// TIA Portal V17 export
// export: Created 2025-03-13T10:29:36.6380281Z, ExportSetting WithDefaults, DisplayName Totally Integrated Automation Portal, DisplayVersion V17 Update 8, DisplayName TIA Portal Openness, DisplayVersion V17 Update 8, DisplayName TIA Portal Version Control Interface, DisplayVersion V17, DisplayName SINAMICS Startdrive Advanced, DisplayVersion V17 SP2, DisplayName SINAMICS Startdrive G110M, G120, G120C, G120D, G120P, G115D, DisplayVersion V17 SP2, DisplayName SINAMICS Startdrive G130, G150, S120, S150, SINAMICS MV, S210, DisplayVersion V17 SP2, DisplayName STEP 7 Professional, DisplayVersion V17 Update 8, DisplayName SINUMERIK ONE STEP 7 Toolbox, DisplayVersion V17 Update 12, DisplayName SINUMERIK 840D sl STEP 7 Toolbox, DisplayVersion V17 Update 12, DisplayName STEP 7 Safety, DisplayVersion V17 Update 6, DisplayName WinCC Advanced, DisplayVersion V17 Update 8
FUNCTION_BLOCK "FB20300_LASER_GUIDE"   // FB20300, LAD
TITLE = FB20300 LASER GUIDE
{ S7_Optimized_Access := 'FALSE' }
VERSION : 0.1
// stored: AutoNumber false, IsIECCheckEnabled false, SetENOAutomatically false, UDAEnableTagReadback false
   VAR_INPUT
      iCONTROL_ON_DELAYED : Bool;
      iLASER_ACTIVE_LASER_ON : Bool;
      iSTART_MANUAL_REQUEST : Bool;
      iSTART_AUTO_REQUEST : Bool;
      iGUIDE_LASER_IS_ON : Bool;
      iSTOP_MANUAL_REQUEST : Bool;
      iSTOP_AUTO_REQUEST : Bool;
      iHOME_SEQUENCE_RUNNING : Bool;
      iCONTROL_OFF : Bool;
      TEMP : Timer;
   END_VAR
   VAR_OUTPUT
      oLASER_NOT_READY_ALARM : Bool;
      oSEOC_ALARMS : Bool;
      oSwitchoncondition_on : Bool;
      oSwitchoncondition_off : Bool;
      oMotion_Active_Right : Bool;
      oMotion_Active_Left : Bool;
      oLimit_right : Bool;
      oLimit_left : Bool;
      oGUIDE_LASER_ON : Bool;
   END_VAR
   VAR DB_SPECIFIC
      DATA : "LASER GUIDE";
   END_VAR
   VAR_TEMP
      DB_NUMBER : DInt;
   END_VAR
   VAR_TEMP   // added for the SCL form of the ladder/FBD networks
      _w1 : Bool;
      _s5time1 : S5Time;
   END_VAR
BEGIN

NETWORK
TITLE = READ INSTANCE DB NUMBER
      L     DINO;
      +     10#800000;
      T     #DB_NUMBER;

REGION Network 2: START GENERAL CONDITIONS / Start General Conditions
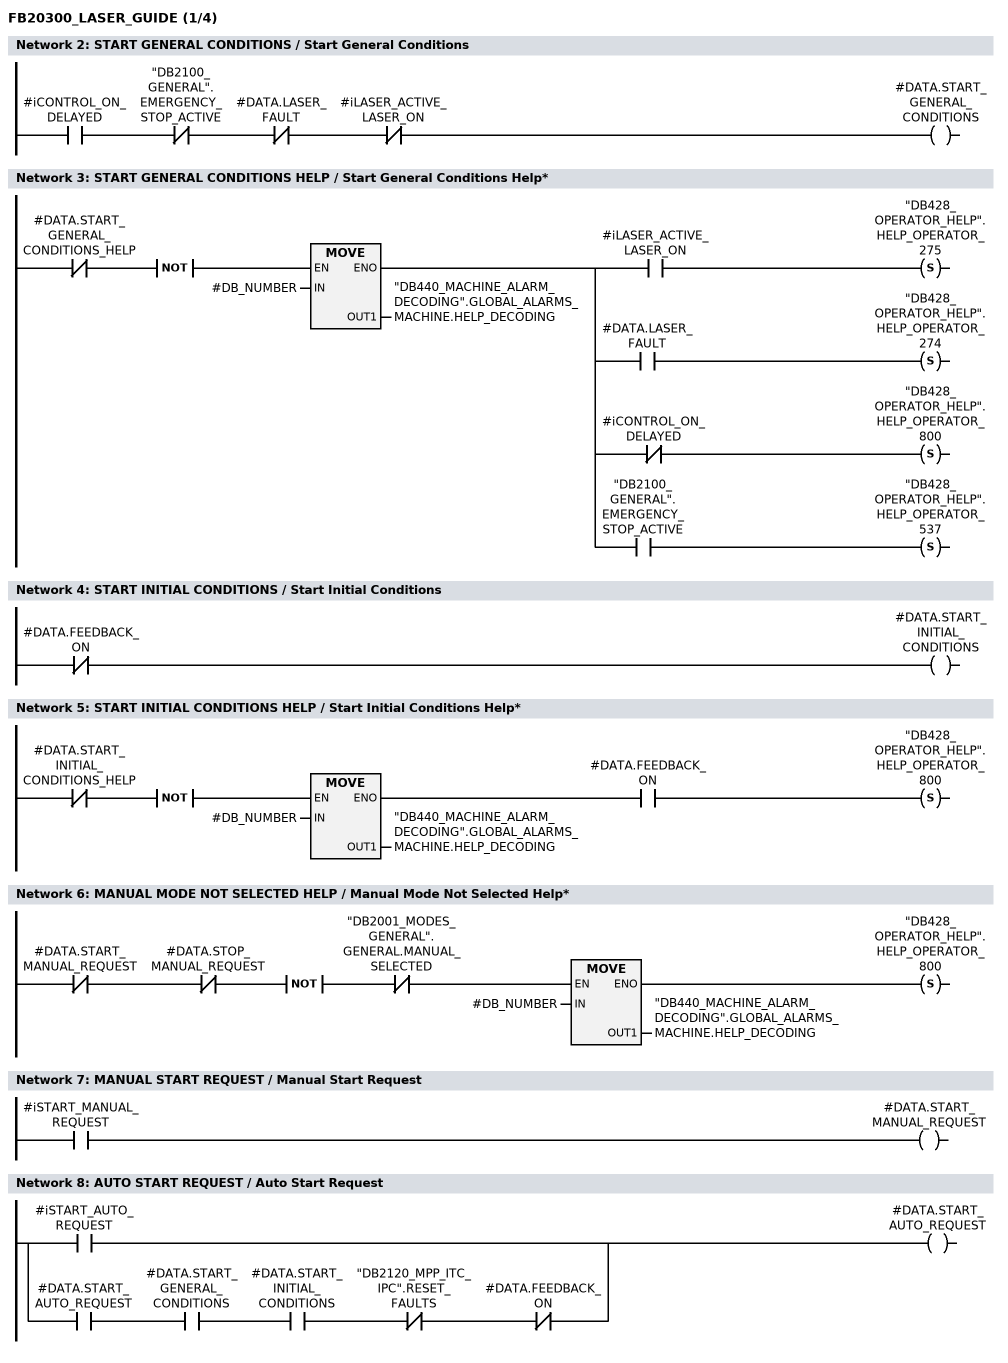
   RUNG wire#powerrail
      Contact( #iCONTROL_ON_DELAYED )
      I_Contact( "DB2100_GENERAL".EMERGENCY_STOP_ACTIVE )
      I_Contact( #DATA.LASER_FAULT )
      I_Contact( #iLASER_ACTIVE_LASER_ON )
      Coil( #DATA.START_GENERAL_CONDITIONS )
   END_RUNG
   // the same network as SCL:
   #DATA.START_GENERAL_CONDITIONS := #iCONTROL_ON_DELAYED AND NOT "DB2100_GENERAL".EMERGENCY_STOP_ACTIVE AND NOT #DATA.LASER_FAULT AND NOT #iLASER_ACTIVE_LASER_ON;
END_REGION

REGION Network 3: START GENERAL CONDITIONS HELP / Start General Conditions Help*
   RUNG wire#powerrail
      I_Contact( #DATA.START_GENERAL_CONDITIONS_HELP )
      Not()
      Move(in := #DB_NUMBER, out1 => "DB440_MACHINE_ALARM_DECODING".GLOBAL_ALARMS_MACHINE.HELP_DECODING)
      wire#w1
      Contact( #iLASER_ACTIVE_LASER_ON )
      S_Coil( "DB428_OPERATOR_HELP".HELP_OPERATOR_275 )
   END_RUNG
   RUNG wire#w1
      Contact( #DATA.LASER_FAULT )
      S_Coil( "DB428_OPERATOR_HELP".HELP_OPERATOR_274 )
   END_RUNG
   RUNG wire#w1
      I_Contact( #iCONTROL_ON_DELAYED )
      S_Coil( "DB428_OPERATOR_HELP".HELP_OPERATOR_800 )
   END_RUNG
   RUNG wire#w1
      Contact( "DB2100_GENERAL".EMERGENCY_STOP_ACTIVE )
      S_Coil( "DB428_OPERATOR_HELP".HELP_OPERATOR_537 )
   END_RUNG
   // the same network as SCL:
   #_w1 := NOT (NOT #DATA.START_GENERAL_CONDITIONS_HELP);
   IF #_w1 THEN "DB440_MACHINE_ALARM_DECODING".GLOBAL_ALARMS_MACHINE.HELP_DECODING := #DB_NUMBER; END_IF;
   IF #_w1 AND #iLASER_ACTIVE_LASER_ON THEN "DB428_OPERATOR_HELP".HELP_OPERATOR_275 := TRUE; END_IF;
   IF #_w1 AND #DATA.LASER_FAULT THEN "DB428_OPERATOR_HELP".HELP_OPERATOR_274 := TRUE; END_IF;
   IF #_w1 AND NOT #iCONTROL_ON_DELAYED THEN "DB428_OPERATOR_HELP".HELP_OPERATOR_800 := TRUE; END_IF;
   IF #_w1 AND "DB2100_GENERAL".EMERGENCY_STOP_ACTIVE THEN
       "DB428_OPERATOR_HELP".HELP_OPERATOR_537 := TRUE;
   END_IF;
END_REGION

REGION Network 4: START INITIAL CONDITIONS / Start Initial Conditions
   RUNG wire#powerrail
      I_Contact( #DATA.FEEDBACK_ON )
      Coil( #DATA.START_INITIAL_CONDITIONS )
   END_RUNG
   // the same network as SCL:
   #DATA.START_INITIAL_CONDITIONS := NOT #DATA.FEEDBACK_ON;
END_REGION

REGION Network 5: START INITIAL CONDITIONS HELP / Start Initial Conditions Help*
   RUNG wire#powerrail
      I_Contact( #DATA.START_INITIAL_CONDITIONS_HELP )
      Not()
      Move(in := #DB_NUMBER, out1 => "DB440_MACHINE_ALARM_DECODING".GLOBAL_ALARMS_MACHINE.HELP_DECODING)
      Contact( #DATA.FEEDBACK_ON )
      S_Coil( "DB428_OPERATOR_HELP".HELP_OPERATOR_800 )
   END_RUNG
   // the same network as SCL:
   #_w1 := NOT (NOT #DATA.START_INITIAL_CONDITIONS_HELP);
   IF #_w1 THEN "DB440_MACHINE_ALARM_DECODING".GLOBAL_ALARMS_MACHINE.HELP_DECODING := #DB_NUMBER; END_IF;
   IF #_w1 AND #DATA.FEEDBACK_ON THEN "DB428_OPERATOR_HELP".HELP_OPERATOR_800 := TRUE; END_IF;
END_REGION

REGION Network 6: MANUAL MODE NOT SELECTED HELP / Manual Mode Not Selected Help*
   RUNG wire#powerrail
      I_Contact( #DATA.START_MANUAL_REQUEST )
      I_Contact( #DATA.STOP_MANUAL_REQUEST )
      Not()
      I_Contact( "DB2001_MODES_GENERAL".GENERAL.MANUAL_SELECTED )
      Move(in := #DB_NUMBER, out1 => "DB440_MACHINE_ALARM_DECODING".GLOBAL_ALARMS_MACHINE.HELP_DECODING)
      S_Coil( "DB428_OPERATOR_HELP".HELP_OPERATOR_800 )
   END_RUNG
   // the same network as SCL:
   IF NOT (NOT #DATA.START_MANUAL_REQUEST AND NOT #DATA.STOP_MANUAL_REQUEST) AND NOT "DB2001_MODES_GENERAL".GENERAL.MANUAL_SELECTED THEN
       "DB440_MACHINE_ALARM_DECODING".GLOBAL_ALARMS_MACHINE.HELP_DECODING := #DB_NUMBER;
       "DB428_OPERATOR_HELP".HELP_OPERATOR_800 := TRUE;
   END_IF;
END_REGION

REGION Network 7: MANUAL START REQUEST / Manual Start Request
   RUNG wire#powerrail
      Contact( #iSTART_MANUAL_REQUEST )
      Coil( #DATA.START_MANUAL_REQUEST )
   END_RUNG
   // the same network as SCL:
   #DATA.START_MANUAL_REQUEST := #iSTART_MANUAL_REQUEST;
END_REGION

REGION Network 8: AUTO START REQUEST / Auto Start Request
   RUNG wire#powerrail
      Contact( #iSTART_AUTO_REQUEST )
      wire#w1
      Coil( #DATA.START_AUTO_REQUEST )
   END_RUNG
   RUNG wire#powerrail
      Contact( #DATA.START_AUTO_REQUEST )
      Contact( #DATA.START_GENERAL_CONDITIONS )
      Contact( #DATA.START_INITIAL_CONDITIONS )
      I_Contact( "DB2120_MPP_ITC_IPC".RESET_FAULTS )
      I_Contact( #DATA.FEEDBACK_ON )
   END_RUNG wire#w1
   // the same network as SCL:
   #DATA.START_AUTO_REQUEST := #iSTART_AUTO_REQUEST OR (#DATA.START_AUTO_REQUEST AND #DATA.START_GENERAL_CONDITIONS AND #DATA.START_INITIAL_CONDITIONS AND NOT "DB2120_MPP_ITC_IPC".RESET_FAULTS AND NOT #DATA.FEEDBACK_ON);
END_REGION

REGION Network 9: START GLOBAL REQUEST / Start Global Request / GLOBAL START REQUEST
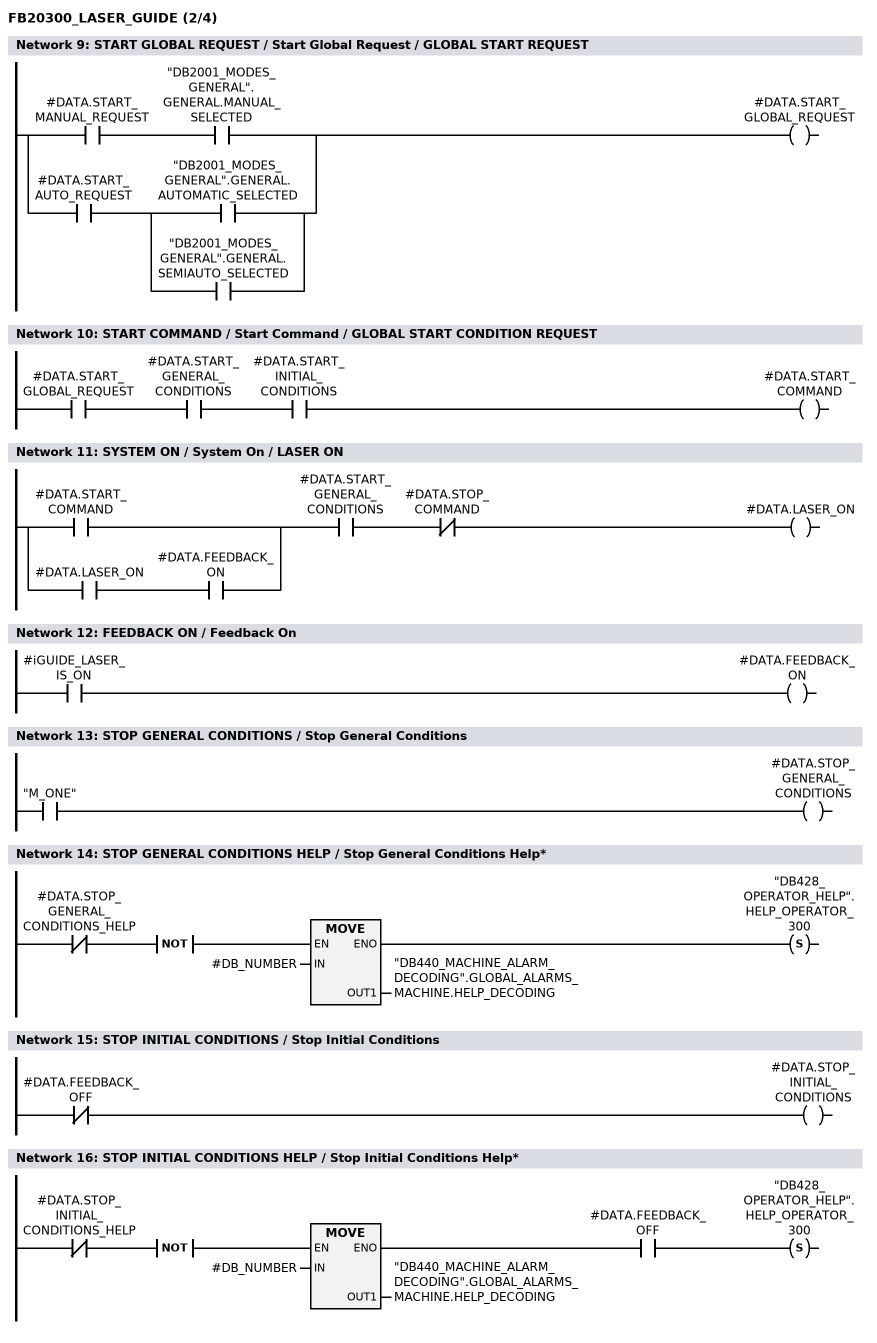
   RUNG wire#powerrail
      Contact( #DATA.START_MANUAL_REQUEST )
      Contact( "DB2001_MODES_GENERAL".GENERAL.MANUAL_SELECTED )
      wire#w1
      Coil( #DATA.START_GLOBAL_REQUEST )
   END_RUNG
   RUNG wire#powerrail
      Contact( #DATA.START_AUTO_REQUEST )
      wire#w2
      Contact( "DB2001_MODES_GENERAL".GENERAL.AUTOMATIC_SELECTED )
   END_RUNG wire#w1
   RUNG wire#w2
      Contact( "DB2001_MODES_GENERAL".GENERAL.SEMIAUTO_SELECTED )
   END_RUNG wire#w1
   // the same network as SCL:
   #DATA.START_GLOBAL_REQUEST := (#DATA.START_MANUAL_REQUEST AND "DB2001_MODES_GENERAL".GENERAL.MANUAL_SELECTED) OR (#DATA.START_AUTO_REQUEST AND ("DB2001_MODES_GENERAL".GENERAL.AUTOMATIC_SELECTED OR "DB2001_MODES_GENERAL".GENERAL.SEMIAUTO_SELECTED));
END_REGION

REGION Network 10: START COMMAND / Start Command / GLOBAL START CONDITION REQUEST
   RUNG wire#powerrail
      Contact( #DATA.START_GLOBAL_REQUEST )
      Contact( #DATA.START_GENERAL_CONDITIONS )
      Contact( #DATA.START_INITIAL_CONDITIONS )
      Coil( #DATA.START_COMMAND )
   END_RUNG
   // the same network as SCL:
   #DATA.START_COMMAND := #DATA.START_GLOBAL_REQUEST AND #DATA.START_GENERAL_CONDITIONS AND #DATA.START_INITIAL_CONDITIONS;
END_REGION

REGION Network 11: SYSTEM ON / System On / LASER ON
   RUNG wire#powerrail
      Contact( #DATA.START_COMMAND )
      wire#w1
      Contact( #DATA.START_GENERAL_CONDITIONS )
      I_Contact( #DATA.STOP_COMMAND )
      Coil( #DATA.LASER_ON )
   END_RUNG
   RUNG wire#powerrail
      Contact( #DATA.LASER_ON )
      Contact( #DATA.FEEDBACK_ON )
   END_RUNG wire#w1
   // the same network as SCL:
   #DATA.LASER_ON := (#DATA.START_COMMAND OR (#DATA.LASER_ON AND #DATA.FEEDBACK_ON)) AND #DATA.START_GENERAL_CONDITIONS AND NOT #DATA.STOP_COMMAND;
END_REGION

REGION Network 12: FEEDBACK ON / Feedback On
   RUNG wire#powerrail
      Contact( #iGUIDE_LASER_IS_ON )
      Coil( #DATA.FEEDBACK_ON )
   END_RUNG
   // the same network as SCL:
   #DATA.FEEDBACK_ON := #iGUIDE_LASER_IS_ON;
END_REGION

REGION Network 13: STOP GENERAL CONDITIONS / Stop General Conditions
   RUNG wire#powerrail
      Contact( "M_ONE" )
      Coil( #DATA.STOP_GENERAL_CONDITIONS )
   END_RUNG
   // the same network as SCL:
   #DATA.STOP_GENERAL_CONDITIONS := "M_ONE";
END_REGION

REGION Network 14: STOP GENERAL CONDITIONS HELP / Stop General Conditions Help*
   RUNG wire#powerrail
      I_Contact( #DATA.STOP_GENERAL_CONDITIONS_HELP )
      Not()
      Move(in := #DB_NUMBER, out1 => "DB440_MACHINE_ALARM_DECODING".GLOBAL_ALARMS_MACHINE.HELP_DECODING)
      S_Coil( "DB428_OPERATOR_HELP".HELP_OPERATOR_300 )
   END_RUNG
   // the same network as SCL:
   IF NOT (NOT #DATA.STOP_GENERAL_CONDITIONS_HELP) THEN
       "DB440_MACHINE_ALARM_DECODING".GLOBAL_ALARMS_MACHINE.HELP_DECODING := #DB_NUMBER;
       "DB428_OPERATOR_HELP".HELP_OPERATOR_300 := TRUE;
   END_IF;
END_REGION

REGION Network 15: STOP INITIAL CONDITIONS / Stop Initial Conditions
   RUNG wire#powerrail
      I_Contact( #DATA.FEEDBACK_OFF )
      Coil( #DATA.STOP_INITIAL_CONDITIONS )
   END_RUNG
   // the same network as SCL:
   #DATA.STOP_INITIAL_CONDITIONS := NOT #DATA.FEEDBACK_OFF;
END_REGION

REGION Network 16: STOP INITIAL CONDITIONS HELP / Stop Initial Conditions Help*
   RUNG wire#powerrail
      I_Contact( #DATA.STOP_INITIAL_CONDITIONS_HELP )
      Not()
      Move(in := #DB_NUMBER, out1 => "DB440_MACHINE_ALARM_DECODING".GLOBAL_ALARMS_MACHINE.HELP_DECODING)
      Contact( #DATA.FEEDBACK_OFF )
      S_Coil( "DB428_OPERATOR_HELP".HELP_OPERATOR_300 )
   END_RUNG
   // the same network as SCL:
   #_w1 := NOT (NOT #DATA.STOP_INITIAL_CONDITIONS_HELP);
   IF #_w1 THEN "DB440_MACHINE_ALARM_DECODING".GLOBAL_ALARMS_MACHINE.HELP_DECODING := #DB_NUMBER; END_IF;
   IF #_w1 AND #DATA.FEEDBACK_OFF THEN "DB428_OPERATOR_HELP".HELP_OPERATOR_300 := TRUE; END_IF;
END_REGION

REGION Network 17: MANUAL STOP REQUEST / Manual Stop Request
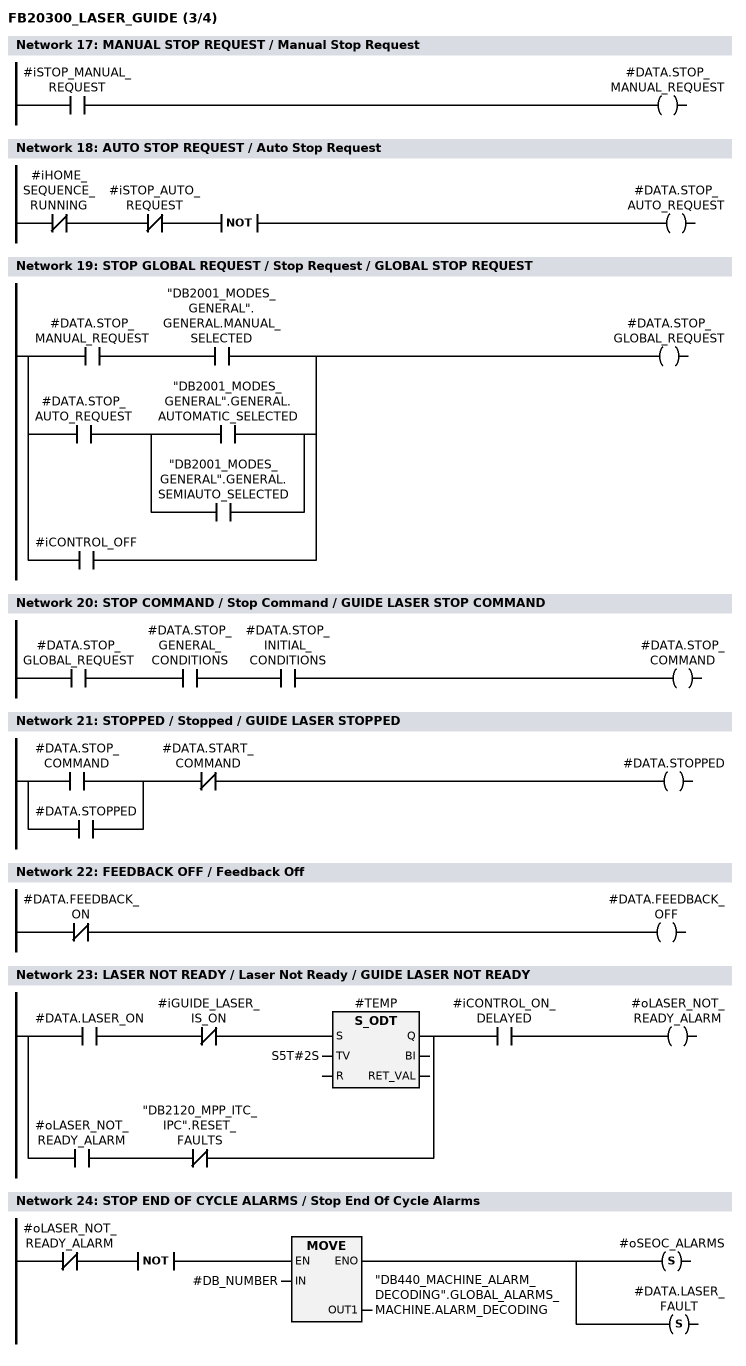
   RUNG wire#powerrail
      Contact( #iSTOP_MANUAL_REQUEST )
      Coil( #DATA.STOP_MANUAL_REQUEST )
   END_RUNG
   // the same network as SCL:
   #DATA.STOP_MANUAL_REQUEST := #iSTOP_MANUAL_REQUEST;
END_REGION

REGION Network 18: AUTO STOP REQUEST / Auto Stop Request
   RUNG wire#powerrail
      I_Contact( #iHOME_SEQUENCE_RUNNING )
      I_Contact( #iSTOP_AUTO_REQUEST )
      Not()
      Coil( #DATA.STOP_AUTO_REQUEST )
   END_RUNG
   // the same network as SCL:
   #DATA.STOP_AUTO_REQUEST := NOT (NOT #iHOME_SEQUENCE_RUNNING AND NOT #iSTOP_AUTO_REQUEST);
END_REGION

REGION Network 19: STOP GLOBAL REQUEST / Stop Request / GLOBAL STOP REQUEST
   RUNG wire#powerrail
      Contact( #DATA.STOP_MANUAL_REQUEST )
      Contact( "DB2001_MODES_GENERAL".GENERAL.MANUAL_SELECTED )
      wire#w1
      Coil( #DATA.STOP_GLOBAL_REQUEST )
   END_RUNG
   RUNG wire#powerrail
      Contact( #DATA.STOP_AUTO_REQUEST )
      wire#w2
      Contact( "DB2001_MODES_GENERAL".GENERAL.AUTOMATIC_SELECTED )
   END_RUNG wire#w1
   RUNG wire#w2
      Contact( "DB2001_MODES_GENERAL".GENERAL.SEMIAUTO_SELECTED )
   END_RUNG wire#w1
   RUNG wire#powerrail
      Contact( #iCONTROL_OFF )
   END_RUNG wire#w1
   // the same network as SCL:
   #DATA.STOP_GLOBAL_REQUEST := (#DATA.STOP_MANUAL_REQUEST AND "DB2001_MODES_GENERAL".GENERAL.MANUAL_SELECTED) OR (#DATA.STOP_AUTO_REQUEST AND ("DB2001_MODES_GENERAL".GENERAL.AUTOMATIC_SELECTED OR "DB2001_MODES_GENERAL".GENERAL.SEMIAUTO_SELECTED)) OR #iCONTROL_OFF;
END_REGION

REGION Network 20: STOP COMMAND / Stop Command / GUIDE LASER STOP COMMAND
   RUNG wire#powerrail
      Contact( #DATA.STOP_GLOBAL_REQUEST )
      Contact( #DATA.STOP_GENERAL_CONDITIONS )
      Contact( #DATA.STOP_INITIAL_CONDITIONS )
      Coil( #DATA.STOP_COMMAND )
   END_RUNG
   // the same network as SCL:
   #DATA.STOP_COMMAND := #DATA.STOP_GLOBAL_REQUEST AND #DATA.STOP_GENERAL_CONDITIONS AND #DATA.STOP_INITIAL_CONDITIONS;
END_REGION

REGION Network 21: STOPPED / Stopped / GUIDE LASER STOPPED
   RUNG wire#powerrail
      Contact( #DATA.STOP_COMMAND )
      wire#w1
      I_Contact( #DATA.START_COMMAND )
      Coil( #DATA.STOPPED )
   END_RUNG
   RUNG wire#powerrail
      Contact( #DATA.STOPPED )
   END_RUNG wire#w1
   // the same network as SCL:
   #DATA.STOPPED := (#DATA.STOP_COMMAND OR #DATA.STOPPED) AND NOT #DATA.START_COMMAND;
END_REGION

REGION Network 22: FEEDBACK OFF / Feedback Off
   RUNG wire#powerrail
      I_Contact( #DATA.FEEDBACK_ON )
      Coil( #DATA.FEEDBACK_OFF )
   END_RUNG
   // the same network as SCL:
   #DATA.FEEDBACK_OFF := NOT #DATA.FEEDBACK_ON;
END_REGION

REGION Network 23: LASER NOT READY / Laser Not Ready / GUIDE LASER NOT READY
   RUNG wire#powerrail
      Contact( #DATA.LASER_ON )
      I_Contact( #iGUIDE_LASER_IS_ON )
      S_ODT(T_NO := #TEMP, TV := S5T#2S, R :=, BI =>, RET_VAL =>)
      wire#w1
      Contact( #iCONTROL_ON_DELAYED )
      Coil( #oLASER_NOT_READY_ALARM )
   END_RUNG
   RUNG wire#powerrail
      Contact( #oLASER_NOT_READY_ALARM )
      I_Contact( "DB2120_MPP_ITC_IPC".RESET_FAULTS )
   END_RUNG wire#w1
   // the same network as SCL:
   #_s5time1 := S_ODT(T_NO := #TEMP, S := #DATA.LASER_ON AND NOT #iGUIDE_LASER_IS_ON, TV := S5T#2S, Q => #_w1);
   #oLASER_NOT_READY_ALARM := (#_w1 OR (#oLASER_NOT_READY_ALARM AND NOT "DB2120_MPP_ITC_IPC".RESET_FAULTS)) AND #iCONTROL_ON_DELAYED;
END_REGION

REGION Network 24: STOP END OF CYCLE ALARMS / Stop End Of Cycle Alarms
   RUNG wire#powerrail
      I_Contact( #oLASER_NOT_READY_ALARM )
      Not()
      Move(in := #DB_NUMBER, out1 => "DB440_MACHINE_ALARM_DECODING".GLOBAL_ALARMS_MACHINE.ALARM_DECODING)
      wire#w1
      S_Coil( #oSEOC_ALARMS )
   END_RUNG
   RUNG wire#w1
      S_Coil( #DATA.LASER_FAULT )
   END_RUNG
   // the same network as SCL:
   IF NOT (NOT #oLASER_NOT_READY_ALARM) THEN
       "DB440_MACHINE_ALARM_DECODING".GLOBAL_ALARMS_MACHINE.ALARM_DECODING := #DB_NUMBER;
       #oSEOC_ALARMS := TRUE;
       #DATA.LASER_FAULT := TRUE;
   END_IF;
END_REGION

REGION Network 25: RESET LASER FAULTED / Reset Laser Faulted / LASER SYSTEM FAULT
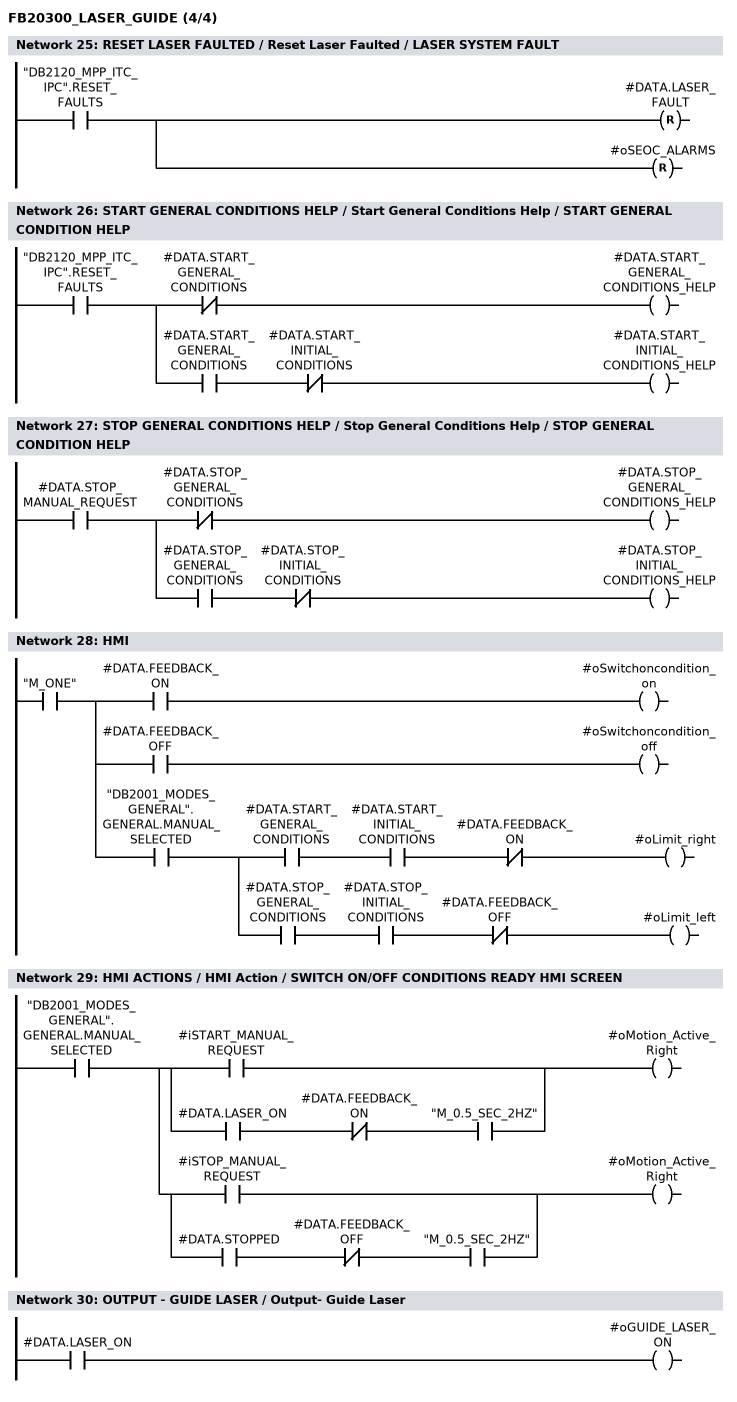
   RUNG wire#powerrail
      Contact( "DB2120_MPP_ITC_IPC".RESET_FAULTS )
      wire#w1
      R_Coil( #DATA.LASER_FAULT )
   END_RUNG
   RUNG wire#w1
      R_Coil( #oSEOC_ALARMS )
   END_RUNG
   // the same network as SCL:
   IF "DB2120_MPP_ITC_IPC".RESET_FAULTS THEN
       #DATA.LASER_FAULT := FALSE;
       #oSEOC_ALARMS := FALSE;
   END_IF;
END_REGION

REGION Network 26: START GENERAL CONDITIONS HELP / Start General Conditions Help / START GENERAL CONDITION HELP
   RUNG wire#powerrail
      Contact( "DB2120_MPP_ITC_IPC".RESET_FAULTS )
      wire#w1
      I_Contact( #DATA.START_GENERAL_CONDITIONS )
      Coil( #DATA.START_GENERAL_CONDITIONS_HELP )
   END_RUNG
   RUNG wire#w1
      Contact( #DATA.START_GENERAL_CONDITIONS )
      I_Contact( #DATA.START_INITIAL_CONDITIONS )
      Coil( #DATA.START_INITIAL_CONDITIONS_HELP )
   END_RUNG
   // the same network as SCL:
   #DATA.START_GENERAL_CONDITIONS_HELP := "DB2120_MPP_ITC_IPC".RESET_FAULTS AND NOT #DATA.START_GENERAL_CONDITIONS;
   #DATA.START_INITIAL_CONDITIONS_HELP := "DB2120_MPP_ITC_IPC".RESET_FAULTS AND #DATA.START_GENERAL_CONDITIONS AND NOT #DATA.START_INITIAL_CONDITIONS;
END_REGION

REGION Network 27: STOP GENERAL CONDITIONS HELP / Stop General Conditions Help / STOP GENERAL CONDITION HELP
   RUNG wire#powerrail
      Contact( #DATA.STOP_MANUAL_REQUEST )
      wire#w1
      I_Contact( #DATA.STOP_GENERAL_CONDITIONS )
      Coil( #DATA.STOP_GENERAL_CONDITIONS_HELP )
   END_RUNG
   RUNG wire#w1
      Contact( #DATA.STOP_GENERAL_CONDITIONS )
      I_Contact( #DATA.STOP_INITIAL_CONDITIONS )
      Coil( #DATA.STOP_INITIAL_CONDITIONS_HELP )
   END_RUNG
   // the same network as SCL:
   #DATA.STOP_GENERAL_CONDITIONS_HELP := #DATA.STOP_MANUAL_REQUEST AND NOT #DATA.STOP_GENERAL_CONDITIONS;
   #DATA.STOP_INITIAL_CONDITIONS_HELP := #DATA.STOP_MANUAL_REQUEST AND #DATA.STOP_GENERAL_CONDITIONS AND NOT #DATA.STOP_INITIAL_CONDITIONS;
END_REGION

REGION Network 28: HMI
   RUNG wire#powerrail
      Contact( "M_ONE" )
      wire#w1
      Contact( #DATA.FEEDBACK_ON )
      Coil( #oSwitchoncondition_on )
   END_RUNG
   RUNG wire#w1
      Contact( #DATA.FEEDBACK_OFF )
      Coil( #oSwitchoncondition_off )
   END_RUNG
   RUNG wire#w1
      Contact( "DB2001_MODES_GENERAL".GENERAL.MANUAL_SELECTED )
      wire#w2
      Contact( #DATA.START_GENERAL_CONDITIONS )
      Contact( #DATA.START_INITIAL_CONDITIONS )
      I_Contact( #DATA.FEEDBACK_ON )
      Coil( #oLimit_right )
   END_RUNG
   RUNG wire#w2
      Contact( #DATA.STOP_GENERAL_CONDITIONS )
      Contact( #DATA.STOP_INITIAL_CONDITIONS )
      I_Contact( #DATA.FEEDBACK_OFF )
      Coil( #oLimit_left )
   END_RUNG
   // the same network as SCL:
   #oSwitchoncondition_on := "M_ONE" AND #DATA.FEEDBACK_ON;
   #oSwitchoncondition_off := "M_ONE" AND #DATA.FEEDBACK_OFF;
   #_w1 := "M_ONE" AND "DB2001_MODES_GENERAL".GENERAL.MANUAL_SELECTED;
   #oLimit_right := #_w1 AND #DATA.START_GENERAL_CONDITIONS AND #DATA.START_INITIAL_CONDITIONS AND NOT #DATA.FEEDBACK_ON;
   #oLimit_left := #_w1 AND #DATA.STOP_GENERAL_CONDITIONS AND #DATA.STOP_INITIAL_CONDITIONS AND NOT #DATA.FEEDBACK_OFF;
END_REGION

REGION Network 29: HMI ACTIONS / HMI Action / SWITCH ON/OFF CONDITIONS READY HMI SCREEN
   RUNG wire#powerrail
      Contact( "DB2001_MODES_GENERAL".GENERAL.MANUAL_SELECTED )
      wire#w1
      Contact( #iSTART_MANUAL_REQUEST )
      wire#w2
      Coil( #oMotion_Active_Right )
   END_RUNG
   RUNG wire#w1
      Contact( #DATA.LASER_ON )
      I_Contact( #DATA.FEEDBACK_ON )
      Contact( "M_0.5_SEC_2HZ" )
   END_RUNG wire#w2
   RUNG wire#w1
      Contact( #iSTOP_MANUAL_REQUEST )
      wire#w3
      Coil( #oMotion_Active_Right )
   END_RUNG
   RUNG wire#w1
      Contact( #DATA.STOPPED )
      I_Contact( #DATA.FEEDBACK_OFF )
      Contact( "M_0.5_SEC_2HZ" )
   END_RUNG wire#w3
   // the same network as SCL:
   #oMotion_Active_Right := "DB2001_MODES_GENERAL".GENERAL.MANUAL_SELECTED AND (#iSTART_MANUAL_REQUEST OR (#DATA.LASER_ON AND NOT #DATA.FEEDBACK_ON AND "M_0.5_SEC_2HZ"));
   #oMotion_Active_Right := "DB2001_MODES_GENERAL".GENERAL.MANUAL_SELECTED AND (#iSTOP_MANUAL_REQUEST OR (#DATA.STOPPED AND NOT #DATA.FEEDBACK_OFF AND "M_0.5_SEC_2HZ"));
END_REGION

REGION Network 30: OUTPUT - GUIDE LASER / Output- Guide Laser
   RUNG wire#powerrail
      Contact( #DATA.LASER_ON )
      Coil( #oGUIDE_LASER_ON )
   END_RUNG
   // the same network as SCL:
   #oGUIDE_LASER_ON := #DATA.LASER_ON;
END_REGION
END_FUNCTION_BLOCK
